TYPE ST_DriveCtrl :
STRUCT
	bDriveRun:BOOL;
	nDriveAnalog:INT;
END_STRUCT
END_TYPE

(* stored: Version 1.1.0.1, ProductVersion 3.1.4024.15
   DUT ST_DriveCtrl: Id {a698a894-8b26-4298-9a14-19409de2033b} *)
